TYPE NodeHandlerControlStruct :
STRUCT
	stop :BOOL; // stop request for stop after end of cycle
	override :LREAL; // velocity orverride in % [0.0 ... 100.0]
END_STRUCT
END_TYPE

(* stored: Version 1.1.0.1
   DUT NodeHandlerControlStruct: Id {fa421bdc-c033-4c17-b866-89326cb2c29d} *)
